TYPE ST_CAMERA_IN :
STRUCT
	stTriggerID			: ST_CAMERA_TriggerID;	
	stBrowserStatus		: ST_CAMERA_BrowserStatus;
	
END_STRUCT
END_TYPE

(* stored: Version 1.1.0.1
   DUT ST_CAMERA_IN: Id {cfbfb277-6114-4e03-9941-c3d926af33b0} *)
